PROGRAM AutoOriginCtrl
VAR
	bDoorHomingBit: BOOL;
	delaystn1move: TON;
	delaystn10move: TON;
	delaySlowpullDownmove: TON;
	delayarm1upmove: TON;
	delayarm2upmove: TON;

	bArm1PnpBusyFE: F_TRIG;
	bAutoStartRE : R_TRIG;
	bTrackerStEnFE: F_TRIG;
	bArm2Stn6PickTo: BOOL;
	bArm2PnpBusyFE: F_TRIG;

	bDoorOriginStep1: BOOL;
	bDoorOriginStep2 : BOOL;
	bDoorOriginStep3: BOOL;
	bDoorOriginStep4: BOOL;
	bDoorOriginStep5: BOOL;
	bDoorOriginStep6: BOOL;
	bDoorOriginStep7: BOOL;
	bDoorOriginStep8: BOOL;

	ARtStnDoorOpenDelayOff: ARRAY [1..iStnQty] OF TON;
	ARtUldDoorOpenDelayOff: TON;
	ARtUldConveyorOpenDelayOff: TON;	

END_VAR
VAR // added by the converter: edge detectors and wires of the graphical bodies
    _w1 : BOOL;
END_VAR

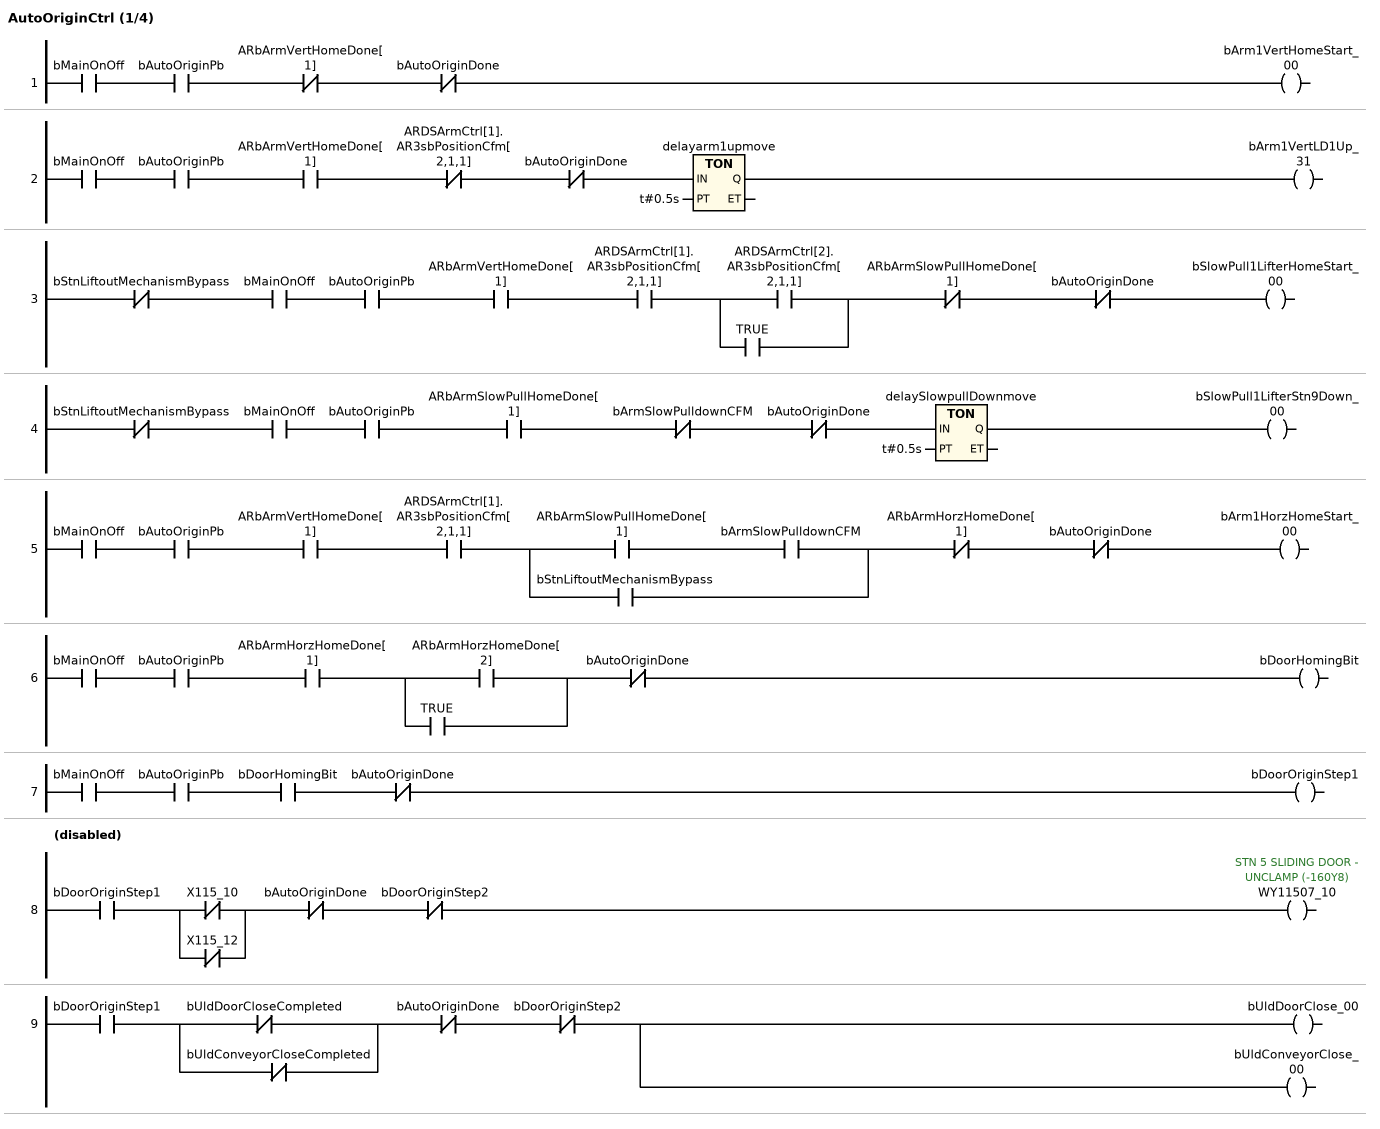
// NETWORK 1
bArm1VertHomeStart_00 := bMainOnOff AND bAutoOriginPb AND NOT ARbArmVertHomeDone[1] AND NOT bAutoOriginDone;

// NETWORK 2
delayarm1upmove(IN := bMainOnOff AND bAutoOriginPb AND ARbArmVertHomeDone[1] AND NOT ARDSArmCtrl[1].AR3sbPositionCfm[2,1,1] AND NOT bAutoOriginDone, PT := t#0.5s); // TON
bArm1VertLD1Up_31 := delayarm1upmove.Q;

// NETWORK 3
bSlowPull1LifterHomeStart_00 := NOT bStnLiftoutMechanismBypass AND bMainOnOff AND bAutoOriginPb AND ARbArmVertHomeDone[1] AND ARDSArmCtrl[1].AR3sbPositionCfm[2,1,1] AND (ARDSArmCtrl[2].AR3sbPositionCfm[2,1,1] OR TRUE) AND NOT ARbArmSlowPullHomeDone[1] AND NOT bAutoOriginDone;

// NETWORK 4
delaySlowpullDownmove(IN := NOT bStnLiftoutMechanismBypass AND bMainOnOff AND bAutoOriginPb AND ARbArmSlowPullHomeDone[1] AND NOT bArmSlowPulldownCFM AND NOT bAutoOriginDone, PT := t#0.5s); // TON
bSlowPull1LifterStn9Down_00 := delaySlowpullDownmove.Q;

// NETWORK 5
bArm1HorzHomeStart_00 := bMainOnOff AND bAutoOriginPb AND ARbArmVertHomeDone[1] AND ARDSArmCtrl[1].AR3sbPositionCfm[2,1,1] AND (ARbArmSlowPullHomeDone[1] AND bArmSlowPulldownCFM OR bStnLiftoutMechanismBypass) AND NOT ARbArmHorzHomeDone[1] AND NOT bAutoOriginDone;

// NETWORK 6
bDoorHomingBit := bMainOnOff AND bAutoOriginPb AND ARbArmHorzHomeDone[1] AND (ARbArmHorzHomeDone[2] OR TRUE) AND NOT bAutoOriginDone;

// NETWORK 7
bDoorOriginStep1 := bMainOnOff AND bAutoOriginPb AND bDoorHomingBit AND NOT bAutoOriginDone;

// NETWORK 8 (disabled)
//   WY11507_10: STN 5 SLIDING DOOR - UNCLAMP (-160Y8)
// WY11507_10 := (bDoorOriginStep1 AND (NOT X115_10 OR NOT X115_12)) AND NOT bAutoOriginDone AND NOT bDoorOriginStep2;

// NETWORK 9
_w1 := bDoorOriginStep1 AND (NOT bUldDoorCloseCompleted OR NOT bUldConveyorCloseCompleted) AND NOT bAutoOriginDone AND NOT bDoorOriginStep2;
bUldDoorClose_00 := _w1;
bUldConveyorClose_00 := _w1;

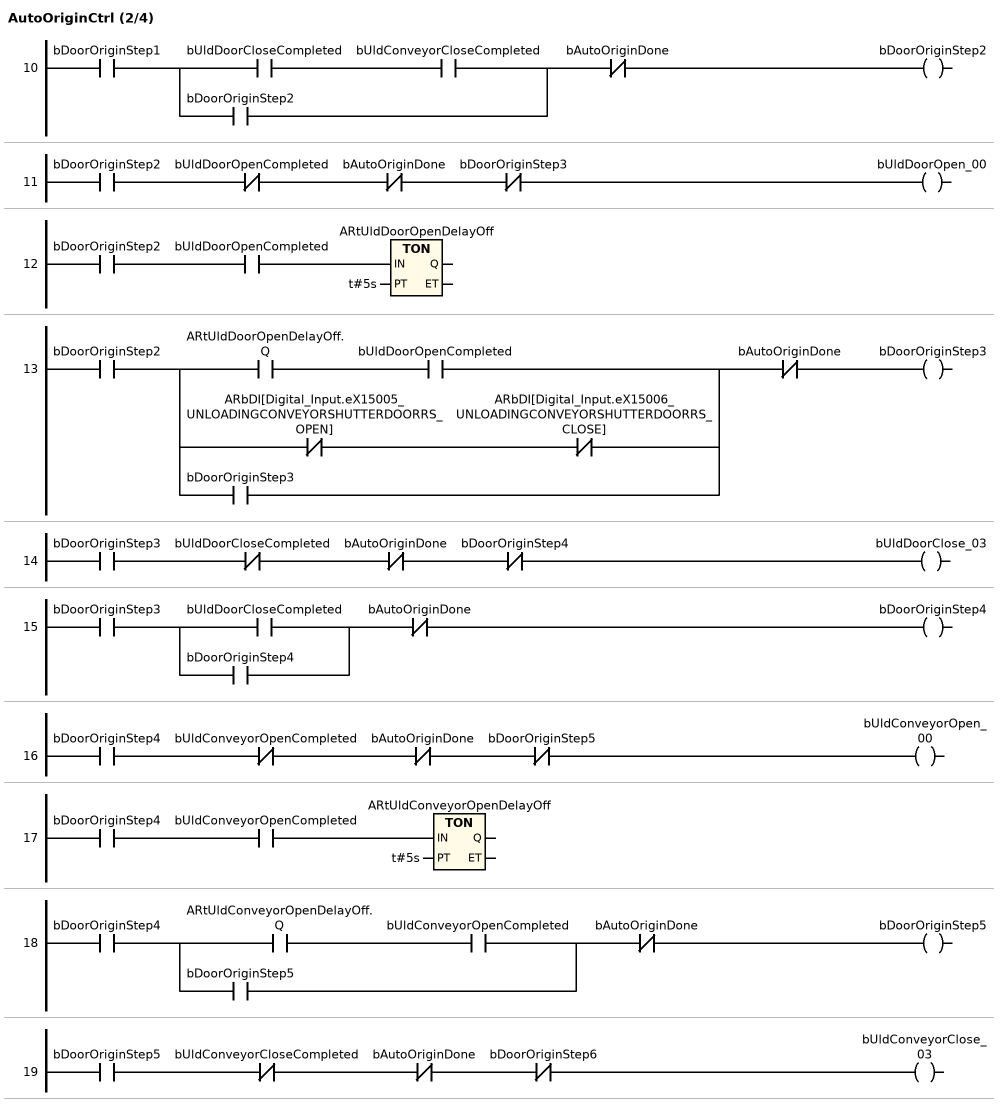
// NETWORK 10
bDoorOriginStep2 := bDoorOriginStep1 AND (bUldDoorCloseCompleted AND bUldConveyorCloseCompleted OR bDoorOriginStep2) AND NOT bAutoOriginDone;

// NETWORK 11
bUldDoorOpen_00 := bDoorOriginStep2 AND NOT bUldDoorOpenCompleted AND NOT bAutoOriginDone AND NOT bDoorOriginStep3;

// NETWORK 12
ARtUldDoorOpenDelayOff(IN := bDoorOriginStep2 AND bUldDoorOpenCompleted, PT := t#5s); // TON

// NETWORK 13
bDoorOriginStep3 := bDoorOriginStep2 AND (ARtUldDoorOpenDelayOff.Q AND bUldDoorOpenCompleted OR NOT ARbDI[Digital_Input.eX15005_UNLOADINGCONVEYORSHUTTERDOORRS_OPEN] AND NOT ARbDI[Digital_Input.eX15006_UNLOADINGCONVEYORSHUTTERDOORRS_CLOSE] OR bDoorOriginStep3) AND NOT bAutoOriginDone;

// NETWORK 14
bUldDoorClose_03 := bDoorOriginStep3 AND NOT bUldDoorCloseCompleted AND NOT bAutoOriginDone AND NOT bDoorOriginStep4;

// NETWORK 15
bDoorOriginStep4 := bDoorOriginStep3 AND (bUldDoorCloseCompleted OR bDoorOriginStep4) AND NOT bAutoOriginDone;

// NETWORK 16
bUldConveyorOpen_00 := bDoorOriginStep4 AND NOT bUldConveyorOpenCompleted AND NOT bAutoOriginDone AND NOT bDoorOriginStep5;

// NETWORK 17
ARtUldConveyorOpenDelayOff(IN := bDoorOriginStep4 AND bUldConveyorOpenCompleted, PT := t#5s); // TON

// NETWORK 18
bDoorOriginStep5 := bDoorOriginStep4 AND (ARtUldConveyorOpenDelayOff.Q AND bUldConveyorOpenCompleted OR bDoorOriginStep5) AND NOT bAutoOriginDone;

// NETWORK 19
bUldConveyorClose_03 := bDoorOriginStep5 AND NOT bUldConveyorCloseCompleted AND NOT bAutoOriginDone AND NOT bDoorOriginStep6;

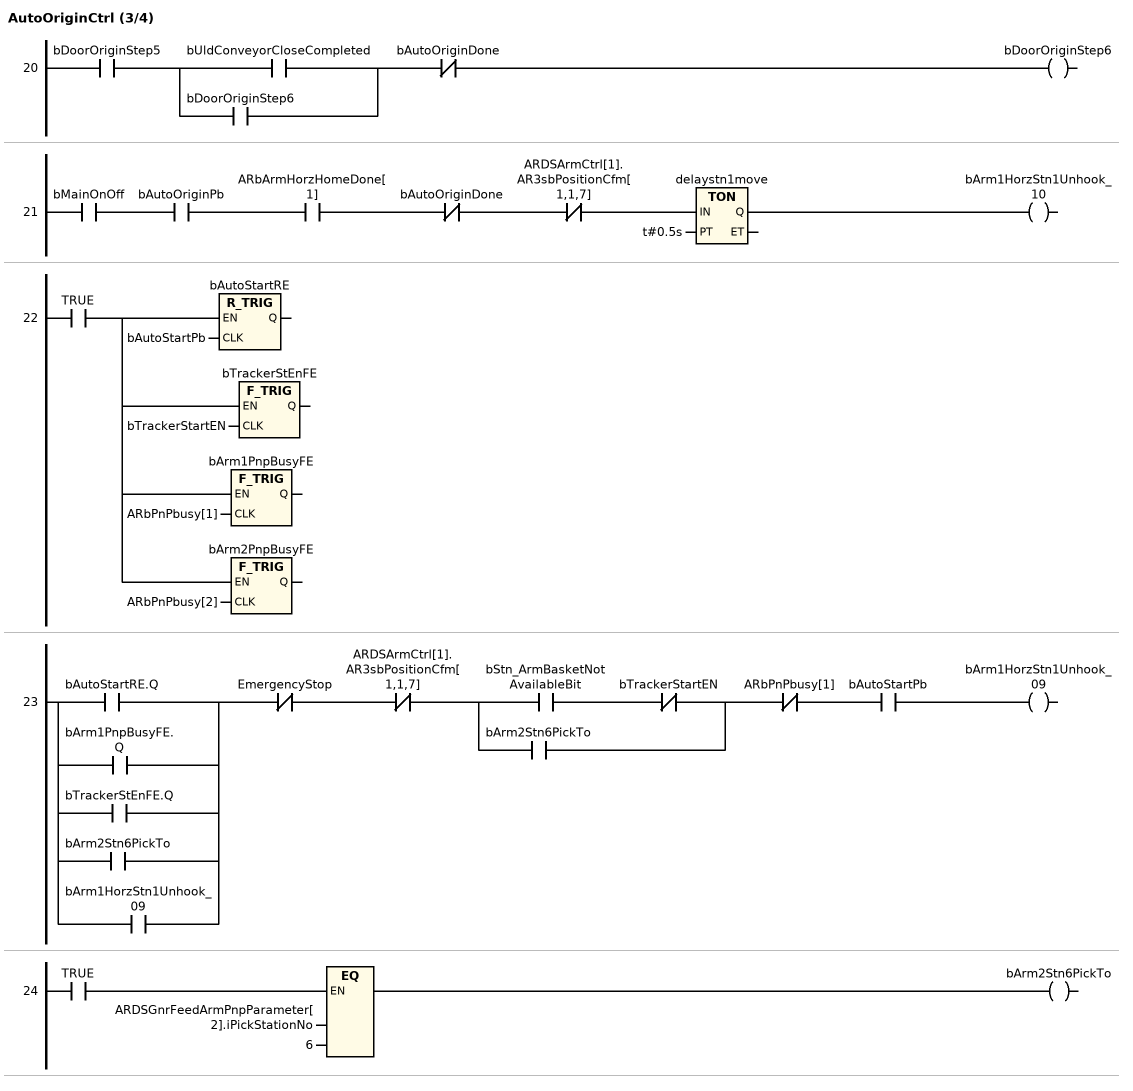
// NETWORK 20
bDoorOriginStep6 := bDoorOriginStep5 AND (bUldConveyorCloseCompleted OR bDoorOriginStep6) AND NOT bAutoOriginDone;

// NETWORK 21
delaystn1move(IN := bMainOnOff AND bAutoOriginPb AND ARbArmHorzHomeDone[1] AND NOT bAutoOriginDone AND NOT ARDSArmCtrl[1].AR3sbPositionCfm[1,1,7], PT := t#0.5s); // TON
bArm1HorzStn1Unhook_10 := delaystn1move.Q;

// NETWORK 22
bAutoStartRE(CLK := bAutoStartPb); // R_TRIG
bTrackerStEnFE(CLK := bTrackerStartEN); // F_TRIG
bArm1PnpBusyFE(CLK := ARbPnPbusy[1]); // F_TRIG
bArm2PnpBusyFE(CLK := ARbPnPbusy[2]); // F_TRIG

// NETWORK 23
bArm1HorzStn1Unhook_09 := ((bAutoStartRE.Q OR bArm1PnpBusyFE.Q OR bTrackerStEnFE.Q OR bArm2Stn6PickTo OR bArm1HorzStn1Unhook_09) AND NOT EmergencyStop AND NOT ARDSArmCtrl[1].AR3sbPositionCfm[1,1,7] AND (bStn_ArmBasketNotAvailableBit AND NOT bTrackerStartEN OR bArm2Stn6PickTo)) AND NOT ARbPnPbusy[1] AND bAutoStartPb;

// NETWORK 24
bArm2Stn6PickTo := ARDSGnrFeedArmPnpParameter[2].iPickStationNo = 6;

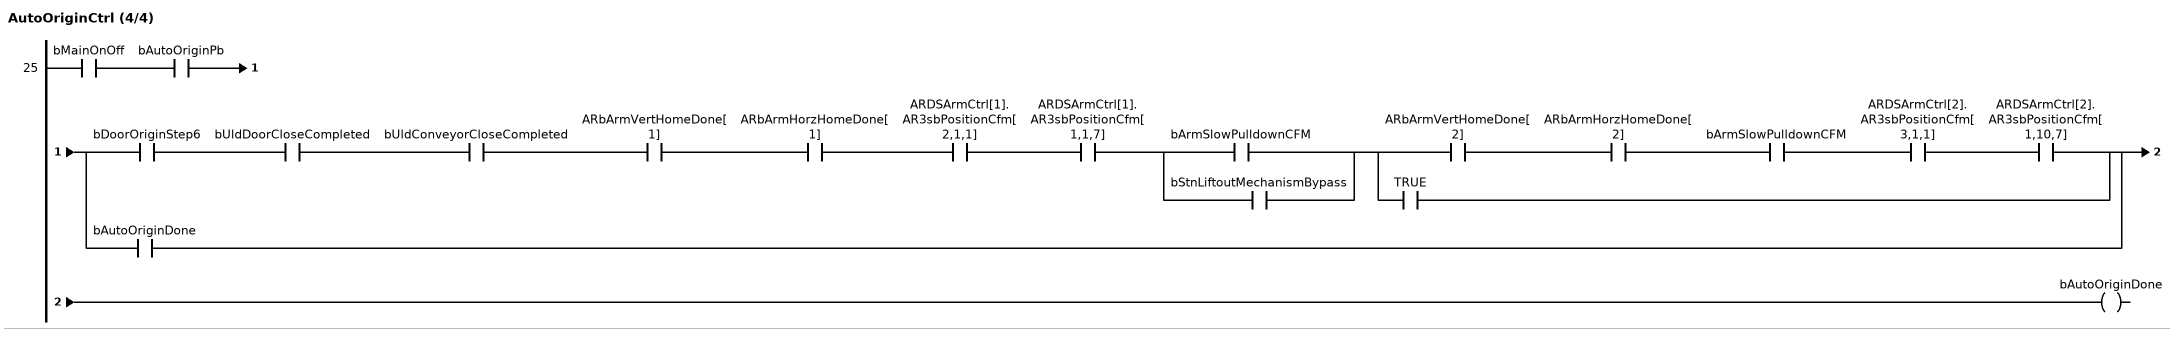
// NETWORK 25
bAutoOriginDone := bMainOnOff AND bAutoOriginPb AND (bDoorOriginStep6 AND bUldDoorCloseCompleted AND bUldConveyorCloseCompleted AND ARbArmVertHomeDone[1] AND ARbArmHorzHomeDone[1] AND ARDSArmCtrl[1].AR3sbPositionCfm[2,1,1] AND ARDSArmCtrl[1].AR3sbPositionCfm[1,1,7] AND (bArmSlowPulldownCFM OR bStnLiftoutMechanismBypass) AND (ARbArmVertHomeDone[2] AND ARbArmHorzHomeDone[2] AND bArmSlowPulldownCFM AND ARDSArmCtrl[2].AR3sbPositionCfm[3,1,1] AND ARDSArmCtrl[2].AR3sbPositionCfm[1,10,7] OR TRUE) OR bAutoOriginDone);

END_PROGRAM

(* stored: Version 1.1.0.1, ProductVersion 3.1.4024.12
   POU AutoOriginCtrl: Id {89a82add-9608-4806-a468-f15f04708de5}, SpecialFunc None *)
